INTERFACE I_HKSystem

END_INTERFACE

(* stored: Version 1.1.0.1, ProductVersion 3.1.4024.12
   Itf I_HKSystem: Id {e28df4ea-6115-43dc-930f-d519283e04cc} *)
